(* IEC 61131-3 sources: AXOpen/src/components.cognex.vision/ctrl/src/AxoVisionPro (part 2) *)

                    IF (Inputs.Status.UserDataLockerJobID = Config.CameraNo) THEN  // IF (Inputs.Status.UserDataLockerJobID = Config.CameraNo) THEN
                        THIS.CallTimers(FALSE);
                        _progress := 384;
                    END_IF;
                END_IF;
                // SendDataTask running: setting the length of the data to sent.
                IF _progress = 384 THEN
                    IF _infoTimer.output THEN
                        TaskMessenger.Activate( UINT#584, eAxoMessageCategory#Potential);
                        Status.Error.Id :=      UINT#584;
                    END_IF;

                    Inputs.Status.WrittenDataVariantSize := _sendDataLength;
                    IF TRUE THEN
                        THIS.CallTimers(FALSE);
                        _progress := 386;
                    END_IF;
                END_IF;
                // SendDataTask running: filling the user data to be sent.
                IF _progress = 386 THEN
                    IF _infoTimer.output THEN
                        TaskMessenger.Activate( UINT#586, eAxoMessageCategory#Potential);
                        Status.Error.Id :=      UINT#586;
                    END_IF;
                    IF _sendDataLength = UINT#0 THEN
                        TaskMessenger.Activate( UINT#1305, eAxoMessageCategory#Error);
                        Status.Error.Id:=       UINT#1305;
                        RETURN;
                    END_IF;
                    //TODO implement error message on the .NET side
                    IF _sendDataLength > UINT#1260 THEN
                        TaskMessenger.Activate( UINT#1308, eAxoMessageCategory#Error);
                        Status.Error.Id:=       UINT#1308;
                        RETURN;
                    END_IF;

                    // Write the user data to the hardware to the UserData_64B_1 'item' from the buffer starting from index 1196.
                    IF _sendDataLength > UINT#1196 THEN
                        _maxindex := System.Math.Min(_sendDataLength - UINT#1, UINT#1263);
                        // Write relevant data from the buffer to the hardware starting from index 1196 in the buffer to index 0 in the hardware.
                        FOR index := UINT#1196 TO _maxindex DO
                            WriteMemory(area := WriteArea#Output,byteOffset := TO_DINT(Config.HWIDs.UserData_64B_1_OutAddress) + TO_DINT(index) - DINT#1196 ,value:= _data_out_1301[index]);
                        END_FOR;
                        // Clear the rest of the hardware buffer after the valid data to avoid sending old data in case of smaller size of data in the next inspections.
                        FOR index := _sendDataLength TO UINT#1263 DO
                            WriteMemory(area := WriteArea#Output,byteOffset := TO_DINT(Config.HWIDs.UserData_64B_1_OutAddress) + TO_DINT(index) - DINT#1196 ,value:= BYTE#0);
                        END_FOR;
                    ELSE
                        // If the data to send is smaller than 1196, clear completelly the hardware buffer.
                        FOR index := UINT#0 TO  UINT#63 DO
                            WriteMemory(area := WriteArea#Output,byteOffset := TO_DINT(Config.HWIDs.UserData_64B_1_OutAddress) + TO_DINT(index),value:= BYTE#0);
                        END_FOR;
                    END_IF;
                    // Write the user data to the hardware to the UserData_240B_5 'item' from the buffer starting from index 956.
                    IF _sendDataLength > UINT#956 THEN
                        _maxindex := System.Math.Min(_sendDataLength - UINT#1, UINT#1195);
                        // Write relevant data from the buffer to the hardware starting from index 956 in the buffer to index 0 in the hardware.
                        FOR index := UINT#956 TO _maxindex DO
                            WriteMemory(area := WriteArea#Output,byteOffset := TO_DINT(Config.HWIDs.UserData_240B_5_OutAddress) + TO_DINT(index) - DINT#956 ,value:= _data_out_1301[index]);
                        END_FOR;
                        // Clear the rest of the hardware buffer after the valid data to avoid sending old data in case of smaller size of data in the next inspections.
                        FOR index := _sendDataLength TO UINT#1195 DO
                            WriteMemory(area := WriteArea#Output,byteOffset := TO_DINT(Config.HWIDs.UserData_240B_5_OutAddress) + TO_DINT(index) - DINT#956 ,value:= BYTE#0);
                        END_FOR;
                    ELSE
                        // If the data to send is smaller than 956, clear completelly the hardware buffer.
                        FOR index := UINT#0 TO  UINT#239 DO
                            WriteMemory(area := WriteArea#Output,byteOffset := TO_DINT(Config.HWIDs.UserData_240B_5_OutAddress) + TO_DINT(index),value:= BYTE#0);
                        END_FOR;
                    END_IF;
                    // Write the user data to the hardware to the UserData_240B_4 'item' from the buffer starting from index 716.
                    IF _sendDataLength > UINT#716 THEN
                        _maxindex := System.Math.Min(_sendDataLength - UINT#1, UINT#955);
                        // Write relevant data from the buffer to the hardware starting from index 716 in the buffer to index 0 in the hardware.
                        FOR index := UINT#716 TO _maxindex DO
                            WriteMemory(area := WriteArea#Output,byteOffset := TO_DINT(Config.HWIDs.UserData_240B_4_OutAddress) + TO_DINT(index) - DINT#716 ,value:= _data_out_1301[index]);
                        END_FOR;
                        // Clear the rest of the hardware buffer after the valid data to avoid sending old data in case of smaller size of data in the next inspections.
                        FOR index := _sendDataLength TO UINT#955 DO
                            WriteMemory(area := WriteArea#Output,byteOffset := TO_DINT(Config.HWIDs.UserData_240B_4_OutAddress) + TO_DINT(index) - DINT#716 ,value:= BYTE#0);
                        END_FOR;
                    ELSE
                        // If the data to send is smaller than 716, clear completelly the hardware buffer.
                        FOR index := UINT#0 TO  UINT#239 DO
                            WriteMemory(area := WriteArea#Output,byteOffset := TO_DINT(Config.HWIDs.UserData_240B_4_OutAddress) + TO_DINT(index),value:= BYTE#0);
                        END_FOR;
                    END_IF;
                    // Write the user data to the hardware to the UserData_240B_3 'item' from the buffer starting from index 476.
                    IF _sendDataLength > UINT#476 THEN
                        _maxindex := System.Math.Min(_sendDataLength - UINT#1, UINT#715);
                        // Write relevant data from the buffer to the hardware starting from index 476 in the buffer to index 0 in the hardware.
                        FOR index := UINT#476 TO _maxindex DO
                            WriteMemory(area := WriteArea#Output,byteOffset := TO_DINT(Config.HWIDs.UserData_240B_3_OutAddress) + TO_DINT(index) - DINT#476 ,value:= _data_out_1301[index]);
                        END_FOR;
                        // Clear the rest of the hardware buffer after the valid data to avoid sending old data in case of smaller size of data in the next inspections.
                        FOR index := _sendDataLength TO UINT#715 DO
                            WriteMemory(area := WriteArea#Output,byteOffset := TO_DINT(Config.HWIDs.UserData_240B_3_OutAddress) + TO_DINT(index) - DINT#476 ,value:= BYTE#0);
                        END_FOR;
                    ELSE
                        // If the data to send is smaller than 476, clear completelly the hardware buffer.
                        FOR index := UINT#0 TO  UINT#239 DO
                            WriteMemory(area := WriteArea#Output,byteOffset := TO_DINT(Config.HWIDs.UserData_240B_3_OutAddress) + TO_DINT(index),value:= BYTE#0);
                        END_FOR;
                    END_IF;
                    // Write the user data to the hardware to the UserData_240B_2 'item' from the buffer starting from index 236.
                    IF _sendDataLength > UINT#236 THEN
                        _maxindex := System.Math.Min(_sendDataLength - UINT#1, UINT#475);
                        // Write relevant data from the buffer to the hardware starting from index 236 in the buffer to index 0 in the hardware.
                        FOR index := UINT#236 TO _maxindex DO
                            WriteMemory(area := WriteArea#Output,byteOffset := TO_DINT(Config.HWIDs.UserData_240B_2_OutAddress) + TO_DINT(index) - DINT#236 ,value:= _data_out_1301[index]);
                        END_FOR;
                        // Clear the rest of the hardware buffer after the valid data to avoid sending old data in case of smaller size of data in the next inspections.
                        FOR index := _sendDataLength TO UINT#475 DO
                            WriteMemory(area := WriteArea#Output,byteOffset := TO_DINT(Config.HWIDs.UserData_240B_2_OutAddress) + TO_DINT(index) - DINT#236 ,value:= BYTE#0);
                        END_FOR;
                    ELSE
                        // If the data to send is smaller than 236, clear completelly the hardware buffer.
                        FOR index := UINT#0 TO  UINT#239 DO
                            WriteMemory(area := WriteArea#Output,byteOffset := TO_DINT(Config.HWIDs.UserData_240B_2_OutAddress) + TO_DINT(index),value:= BYTE#0);
                        END_FOR;
                    END_IF;
                    // Write the user data to the hardware to the UserData_240B_1 'item' from the buffer starting from index 4.
                    IF _sendDataLength > UINT#0 THEN
                        _maxindex := System.Math.Min(_sendDataLength - UINT#1, UINT#235);
                        // Write relevant data from the buffer to the hardware starting from index 0 in the buffer to index 4 in the hardware.
                        FOR index := UINT#0 TO _maxindex DO
                            WriteMemory(area := WriteArea#Output,byteOffset := TO_DINT(Config.HWIDs.UserData_240B_1_OutAddress) + TO_DINT(index) + DINT#4 ,value:= _data_out_1301[index]);
                        END_FOR;
                        // Clear the rest of the hardware buffer after the valid data to avoid sending old data in case of smaller size of data in the next inspections.
                        FOR index := _sendDataLength TO UINT#235 DO
                            WriteMemory(area := WriteArea#Output,byteOffset := TO_DINT(Config.HWIDs.UserData_240B_1_OutAddress) + TO_DINT(index) + DINT#4 ,value:= BYTE#0);
                        END_FOR;
                    ELSE
                        // If the data to send is smaller than 0, clear completelly the hardware buffer.
                        FOR index := UINT#0 TO  UINT#235 DO
                            WriteMemory(area := WriteArea#Output,byteOffset := TO_DINT(Config.HWIDs.UserData_240B_1_OutAddress) + TO_DINT(index) + DINT#4 ,value:= BYTE#0);
                        END_FOR;
                    END_IF;

                    IF TRUE THEN
                        THIS.CallTimers(FALSE);
                        _progress := 387;
                    END_IF;
                END_IF;
                // SendDataTask running: waiting for falling of the set user data acknowledge.
                IF _progress = 387 THEN
                    IF _infoTimer.output THEN
                        TaskMessenger.Activate( UINT#587, eAxoMessageCategory#Potential);
                        Status.Error.Id :=      UINT#587;
                    END_IF;

                    IF NOT Inputs.Status.SetUserDataAck THEN
                        Outputs.Control.SetUserdata := TRUE;
                        THIS.CallTimers(FALSE);
                        _progress := 388;
                    END_IF;
                END_IF;
                // SendDataTask running: waiting for the confirmation of the user data.
                IF _progress = 388 THEN
                    IF _infoTimer.output THEN
                        TaskMessenger.Activate( UINT#588, eAxoMessageCategory#Potential);
                        Status.Error.Id :=      UINT#588;
                    END_IF;

                    IF Inputs.Status.SetUserDataAck THEN
                        Outputs.Control.SetUserdata := FALSE;
                        THIS.CallTimers(FALSE);
                        _progress := 389;
                    END_IF;
                END_IF;
                // SendDataTask running: waiting for falling of the set user data acknowledge.
                IF _progress = 389 THEN
                    IF _infoTimer.output THEN
                        TaskMessenger.Activate( UINT#589, eAxoMessageCategory#Potential);
                        Status.Error.Id :=      UINT#589;
                    END_IF;

                    IF NOT Inputs.Status.SetUserDataAck THEN
                        THIS.CallTimers(FALSE);
                        _progress := 390;
                    END_IF;
                END_IF;
                // SendDataTask running: waiting for falling of the set user data acknowledge.
                IF _progress = 390 THEN
                    IF _infoTimer.output THEN
                        TaskMessenger.Activate( UINT#590, eAxoMessageCategory#Potential);
                        Status.Error.Id :=      UINT#590;
                    END_IF;

                    WriteMemory(area := WriteArea#Output,byteOffset := TO_DINT(Config.HWIDs.UserData_240B_1_OutAddress) + DINT#0,value:= BYTE#0);
                    WriteMemory(area := WriteArea#Output,byteOffset := TO_DINT(Config.HWIDs.UserData_240B_1_OutAddress) + DINT#1,value:= BYTE#0);
                    Outputs.Control.WriteDataId := BYTE#0;

                    IF TRUE THEN
                        THIS.CallTimers(FALSE);
                        _progress := 391;
                    END_IF;
                END_IF;
                // SendDataTask running: data handler set.
                IF _progress = 391 THEN
                    IF _infoTimer.output THEN
                        TaskMessenger.Activate( UINT#591, eAxoMessageCategory#Potential);
                        Status.Error.Id :=      UINT#591;
                    END_IF;

                    IF NOT Inputs.Status.SoftEvent.DataHandlerDone THEN
                        Outputs.Control.SoftEvent.DataHandlerAck := TRUE;
                        THIS.CallTimers(FALSE);
                        _progress := 392;
                    END_IF;
                END_IF;
                // SendDataTask running: waiting for data handler ack.
                IF _progress = 392 THEN
                    IF _infoTimer.output THEN
                        TaskMessenger.Activate( UINT#592, eAxoMessageCategory#Potential);
                        Status.Error.Id :=      UINT#592;
                    END_IF;

                    IF Inputs.Status.SoftEvent.DataHandlerDone THEN
                        Outputs.Control.SoftEvent.DataHandlerAck := FALSE;
                        THIS.CallTimers(FALSE);
                        _progress := 393;
                    END_IF;
                END_IF;
                // SendDataTask running: waiting for data handler ack false.
                IF _progress = 393 THEN
                    IF _infoTimer.output THEN
                        TaskMessenger.Activate( UINT#593, eAxoMessageCategory#Potential);
                        Status.Error.Id :=      UINT#593;
                    END_IF;

                    IF NOT Inputs.Status.SoftEvent.DataHandlerDone THEN
                        THIS.CallTimers(FALSE);
                        _progress := 394;
                    END_IF;
                END_IF;
                // SendDataTask finished.
                IF _progress = 394 THEN
                    SendDataTask.DoneWhen(TRUE);
                    _progress := 0;
                END_IF;

                THIS.CallTimers(TRUE);

                SendDataTask.ThrowWhen(_errorTimer.output);
                Status.Action.Id := TO_UINT(_progress);
                SendDataTask.ThrowWhen(SendDataTask.Duration >= Config.TaskTimeout AND Config.TaskTimeout > T#0s ,'<#SendDataTask timeout.#>');
            END_IF;
            IF SendDataTask.DoneReached() THEN
                Status.Action.Id :=  UINT#181;
                Status.Error.Id :=  UINT#0;
            ELSIF SendDataTask.ErrorOccured() THEN
                Status.Action.Id :=  UINT#10080;
                Status.Error.Id  :=  UINT#10080;
            ELSIF SendDataTask.AbortTriggered()THEN
                Status.Action.Id :=  UINT#10081;
                Status.Error.Id  :=  UINT#10081;
            END_IF;
            Messenger.ActivateOnCondition(ULINT#10080,SendDataTask.HasError(), eAxoMessageCategory#Error);
            Messenger.ActivateOnCondition(ULINT#10081,SendDataTask.IsAborted(), eAxoMessageCategory#Error);
            Messenger.ActivateOnCondition(ULINT#182,SendDataTask.RestoreTriggered() , eAxoMessageCategory#Error);
            IF SendDataTask.RestoreTriggered() AND _progress >= 380 AND _progress <= 399  THEN
                Status.Action.Id :=  UINT#182;
                _progress := 0;
            END_IF;
            //**************************************************

            //***********Update outputs ****************

			IF    CameraNo = BYTE#1 THEN
					_outputsAddress := Config.HWIDs.SystemControl_OutAddress + UDINT#4;
					_bitOffset := 0;
            ELSIF CameraNo = BYTE#2 THEN
					_outputsAddress := Config.HWIDs.SystemControl_OutAddress + UDINT#4;
					_bitOffset := 4;
            ELSIF CameraNo = BYTE#3 THEN
					_outputsAddress := Config.HWIDs.SystemControl_OutAddress + UDINT#5;
					_bitOffset := 0;
            ELSIF CameraNo = BYTE#4 THEN
					_outputsAddress := Config.HWIDs.SystemControl_OutAddress + UDINT#5;
					_bitOffset := 4;
            ELSIF CameraNo = BYTE#5 THEN
					_outputsAddress := Config.HWIDs.SystemControl_OutAddress + UDINT#6;
					_bitOffset := 0;
            ELSIF CameraNo = BYTE#6 THEN
					_outputsAddress := Config.HWIDs.SystemControl_OutAddress + UDINT#6;
					_bitOffset := 4;
            ELSIF CameraNo = BYTE#7 THEN
					_outputsAddress := Config.HWIDs.SystemControl_OutAddress + UDINT#7;
					_bitOffset := 0;
            ELSIF CameraNo = BYTE#8 THEN
					_outputsAddress := Config.HWIDs.SystemControl_OutAddress + UDINT#7;
					_bitOffset := 4;
			END_IF;

			WriteMemory(area := WriteArea#Output,byteOffset := TO_DINT(Config.HWIDs.SystemControl_OutAddress), bitOffset := _bitOffset, value:= Outputs.Control.SoftEvent.Reset);
			WriteMemory(area := WriteArea#Output,byteOffset := TO_DINT(Config.HWIDs.SystemControl_OutAddress), bitOffset := _bitOffset + INT#1, value:= Outputs.Control.SoftEvent.DataHandlerAck);
			WriteMemory(area := WriteArea#Output,byteOffset := TO_DINT(Config.HWIDs.SystemControl_OutAddress), bitOffset := _bitOffset + INT#2, value:= Outputs.Control.SoftEvent.Trigger);
			WriteMemory(area := WriteArea#Output,byteOffset := TO_DINT(Config.HWIDs.SystemControl_OutAddress), bitOffset := _bitOffset + INT#3, value:= Outputs.Control.SoftEvent.Reserve);

			IF (Inputs.Status.ReadDataLockerJobID = Config.CameraNo) THEN
				WriteMemory(area := WriteArea#Output,byteOffset := TO_DINT(Config.HWIDs.SystemControl_OutAddress), bitOffset := INT#4, value:= Outputs.Control.InitiateJobLoad );

				WriteMemory(area := WriteArea#Output,byteOffset := TO_DINT(Config.HWIDs.SystemControl_OutAddress) + DINT#2, value:= Outputs.Control.JobLoadID);

		        WriteMemory(area := WriteArea#Output,byteOffset := TO_DINT(Config.HWIDs.EngineControl_1_OutAddress), bitOffset := INT#1, value:= Outputs.Control.InspectionResultsAck);
			END_IF;

			IF  (Inputs.Status.UserDataLockerJobID = Config.CameraNo) THEN
				WriteMemory(area := WriteArea#Output,byteOffset := TO_DINT(Config.HWIDs.EngineControl_1_OutAddress), bitOffset := INT#3, value:= Outputs.Control.SetUserdata);
			END_IF;

			// -   User Data [20-1400]: Spolocny buffer pre user data. Vyuziva sa vzdy cely buffer (v jednom CASE moze pristupovat len jedna inspekcia).
			//     o   Byte[0]: cislo inspekcie (camera*10 + ( 0 az 9)), pre ktore su aktualne data v bufferi platne
			//     o   Byte[1]: typ spracovania dat (0 = Undefined, 1 = Zmena jobu/referencie, )
			//     o   Byte[2]: cislo jobu
			//     o   Byte[3-??]: id kusu

            //******************************************

        END_METHOD

        METHOD PUBLIC HardResetAllCameras : IAxoTaskState
            HardResetAllCameras := HardResetAllCamerasTask.Invoke(THIS);
        END_METHOD

        METHOD PUBLIC Reset : IAxoTaskState
            Reset := ResetTask.Invoke(THIS);
        END_METHOD

        METHOD PUBLIC Trigger : IAxoTaskState
            Trigger := TriggerTask.Invoke(THIS);
        END_METHOD

        METHOD PUBLIC ReadResults : IAxoTaskState
            VAR_INPUT
                JobID       :   BYTE;
                Length      :   UINT;
            END_VAR
            VAR_IN_OUT
                Data : ARRAY[0..1300] OF BYTE;
            END_VAR
            _readResultsJobID   :=  JobID;
            _readResultsLength  :=  Length;
            Data := _data_in_1301; // copy data to target array
            ReadResults         :=  ReadResultsTask.Invoke(THIS);
        END_METHOD

        METHOD PUBLIC SendData : IAxoTaskState
            VAR_INPUT
                InspectionType  :   BYTE;   // (0 = Undefined, 1 = Zmena jobu/referencie, 2=Nacitanie
                BufferID        :   BYTE;   // Buffer ID, 0-9
                JobID           :   BYTE;
                Length          :   UINT;
            END_VAR
            VAR_IN_OUT
                Data : ARRAY[0..1300] OF BYTE;
            END_VAR
            _sendDataInspectionType :=  InspectionType;
            _sendDataBufferID       :=  BufferID;
            _sendDataJobID          :=  JobID;
            _sendDataLength         :=  Length;
            _data_out_1301          :=  Data;
            SendData                :=  SendDataTask.Invoke(THIS);
        END_METHOD

        METHOD PROTECTED OVERRIDE ManualControl
            THIS._isManuallyControllable := TRUE;

            _readResultsJobID       :=  ReadResultsJobIDServiceMode;
            _readResultsLength      :=  ReadResultsLengthServiceMode;
            _data_in_1301           :=  ResultData.Data;

            _sendDataInspectionType :=  SendDataInspectionTypeServiceMode;
            _sendDataBufferID       :=  SendDataBufferIDServiceMode;
            _sendDataJobID          :=  SendResultsJobIDServiceMode;
            _sendDataLength         :=  SendResultsLengthServiceMode;
            _data_out_1301          :=  UserData.Data;

        END_METHOD

        ///<summary>
        /// Restores this component into intial state.
        ///</summary>
        METHOD PUBLIC OVERRIDE Restore
            VAR
                _index : INT;
            END_VAR
            Status.Action.Id := UINT#0;
            Status.Error.Id  := UINT#0;

            _progress       :=   INT#0;

            FOR _index := 0 TO 1300 DO
                _data_in_1301[_index] := BYTE#0;
                _data_out_1301[_index] := BYTE#0;
            END_FOR;

            HardResetAllCamerasTask.Restore();
            ResetTask.Restore();
            TriggerTask.Restore();
            ReadResultsTask.Restore();
            SendDataTask.Restore();
            HardwareDiagnosticsTask.Restore();

            Status.Action.Id := UINT#50;
            RestoreTask.DoneWhen(TRUE);

        END_METHOD

        METHOD PRIVATE CallTimers
            VAR_INPUT
                signal : BOOL;
            END_VAR

            _infoTimer.OnDelay(THIS, signal AND Config.InfoTime > LT#0S ,Config.InfoTime);
            _errorTimer.OnDelay(THIS, signal AND Config.ErrorTime > LT#0S , Config.ErrorTime);
        END_METHOD

    END_CLASS
END_NAMESPACE
